Staubli VAL3: movel_pulseDO.pgx

public program movel_pulseDO(point x_pPoint, tool x_tTool, mdesc x_mMdesc, dio& x_dDio, num x_nPulseLength)
  local num l_nDist
  local num l_nIndex
  local bool l_bRes
begin

  //execute a movel with the usual arguments (x_pPoint, x_tTool, x_mMdesc) meanwhile
  //when the distance between x_tTool and x_pPoint is lesser than x_nDistance the output x_dDio produce an output of x_nPulseLength seconds

  //the stack is busy
  if bAdvMoves
    l_bRes = watch(!bAdvMoves, nDeadLockTout)
    if !l_bRes
      //it seems stuck!
      call advMovesEmpty(l_bRes)
      //check the "stack" compliance
      call checkAdvMoves()
      if l_bRes
        //but the stack is empty...someone changed it to true manually and saved the library?
        bAdvMoves = false
        libSave()
        logMsg("libSignals/movel_pulseDO->deadlock fixed")
      endIf
    endIf
  endIf

  setMutex(bAdvMoves)

  if x_mMdesc.blend==off
    l_nDist=nBlendOffToll
  else
    l_nDist=x_mMdesc.leave+nBlendOnToll
  endIf

  //check the "stack" compliance
  call checkAdvMoves()

  //get the first index available
  l_nIndex=-1
  while l_nIndex<0
    call avaAdvMoveIndex(l_nIndex)
    delay(0)
  endWhile

  if taskStatus(sAdvMovePrefix+toString("",l_nIndex))==-1
    call lockAdvMove(l_nIndex)
    taskCreate sAdvMovePrefix+toString("",l_nIndex),10,exeMove_pulseDO(l_nIndex, movel(x_pPoint,x_tTool,x_mMdesc),x_pPoint,x_tTool,l_nDist,x_nPulseLength,x_dDio)
    //launch id watchdog
    call launchIdWD()
  else
    logMsg("libSignals/movel_pulseDO->error creating the control task")
  endIf

  bAdvMoves = false


end
